// TIA Portal project "bao_cao" (V15.1)

(* hardware
DEVICE "S71500/ET200MP station_1"  S7-1500 station
   slot 0: "Rail_0"  Rack  6ES7 590-1***0-0AA0
   slot 1: "PLC_1"  CPU 1516-3 PN/DP  6ES7 516-3AN00-0AB0  V1.7
DEVICE "PC-System_1"  SIMATIC PC station
   slot 0: "SIMATIC PC station"  Rail  SIMATIC PC-Station  V1.0
      slot 125: "Stationmanager"  Station_Manager  V6.0.4
   slot 1: "HMI_RT_1"  WinCC RT Advanced  6AV2 104-0xxxx-xxxx  15.1.0.0
      slot 33792: "Host interface"  Host interface
   slot 2: "IE general_1"  IE General  IE_CP  V8.2.0
*)

// ===== PLC "PLC_1"  CPU 1516-3 PN/DP =====

VAR_GLOBAL   // PLC tag table "Default tag table"
   "Tag_1" AT %M100.0 : Bool;
END_VAR

VAR_GLOBAL   // PLC tag table "INPUT"
   "BI_START" AT %I0.0 : Bool;
   "BI_STOP" AT %I0.1 : Bool;
   "BI_AUTO" AT %I0.2 : Bool;
   "BI_MANU" AT %I0.3 : Bool;
   "I_CB1" AT %I0.4 : Bool;
   "I_CB2" AT %I0.5 : Bool;
   "I_CB3" AT %I0.6 : Bool;
   "I_CB_DAY" AT %I0.7 : Bool;
   "BM_START" AT %M0.0 : Bool;
   "BM_STOP" AT %M0.1 : Bool;
   "BM_AUTO" AT %M0.2 : Bool;
   "BM_MANU" AT %M0.3 : Bool;
   "M_CB1" AT %M0.4 : Bool;
   "M_CB2" AT %M0.5 : Bool;
   "M_CB3" AT %M0.6 : Bool;
   "M_CB_DAY" AT %M0.7 : Bool;
   "BM_SIMULATION" AT %M1.0 : Bool;
   "BIT_GIU" AT %M1.1 : Bool;
END_VAR

VAR_GLOBAL   // PLC tag table "OUTPUT"
   "Q_DEN_LV" AT %Q0.0 : Bool;
   "Q_BT" AT %Q0.1 : Bool;
   "Q_BOM_DL" AT %Q0.2 : Bool;
   "Q_XLC1" AT %Q0.3 : Bool;
   "Q_XLC2" AT %Q0.4 : Bool;
   "Q_XLK1" AT %Q0.5 : Bool;
   "Q_XLK2" AT %Q0.6 : Bool;
   "Q_XL_DAY_NAP" AT %Q0.7 : Bool;
   "Q_XL_DONG_NAP" AT %Q1.0 : Bool;
END_VAR

VAR_GLOBAL   // PLC tag table "DEM_SP"
   "DEM_CB1" AT %MW100 : Int;
   "DEM_CB2" AT %MW102 : Int;
   "DEM_CB3" AT %MW104 : Int;
END_VAR

VAR_GLOBAL   // PLC tag table "LENH_P&N"
   "P1" AT %M10.0 : Bool;
   "P2" AT %M10.1 : Bool;
   "BIT_DELAY3S_1" AT %M10.2 : Bool;
   "BIT_DELAY3S_2" AT %M10.3 : Bool;
   "BAO_DANG_ROT" AT %M10.4 : Bool;
   "BAO_DANG_DAP_NAP" AT %M10.5 : Bool;
   "BIT_DELAY3S_3" AT %M10.6 : Bool;
   "BIT_DELAY1S_1" AT %M10.7 : Bool;
   "BIT_DELAY1S_2" AT %M11.0 : Bool;
   "BIT_DELAY3S_4" AT %M11.1 : Bool;
   "BIT_DELAY3S_5" AT %M11.2 : Bool;
   "P3" AT %M11.3 : Bool;
   "P4" AT %M11.4 : Bool;
   "P5" AT %M11.5 : Bool;
   "P6" AT %M11.6 : Bool;
   "P7" AT %M11.7 : Bool;
   "P8" AT %M12.0 : Bool;
   "XUNG_1S" AT %M12.1 : Bool;
   "P10" AT %M12.2 : Bool;
   "P11" AT %M12.3 : Bool;
   "P12" AT %M12.4 : Bool;
   "P13" AT %M12.5 : Bool;
   "P14" AT %M12.6 : Bool;
   "P15" AT %M12.7 : Bool;
   "P16" AT %M13.0 : Bool;
END_VAR

VAR_GLOBAL   // PLC tag table "SIMULATION"
   "SIMU_DOAN_1" AT %MW106 : Int;
   "SIMU_DOAN_2" AT %MW108 : Int;
   "SIMU_DOAN_3" AT %MW110 : Int;
   "BIT_CHAI_MOVE_DOAN_1" AT %M20.0 : Bool;
   "BIT_CHAI_MOVE_DOAN_2" AT %M20.1 : Bool;
   "BIT_CHAI_MOVE_DOAN_3" AT %M20.2 : Bool;
   "SIMU_CHAI_DANG_DONG_NAP" AT %M20.3 : Bool;
   "SIMU_CHAI_DANG_ROT" AT %M20.4 : Bool;
END_VAR

// folder: System blocks/Program resources

DATA_BLOCK "IEC_Timer_0_DB"   // DB1
{ S7_Optimized_Access := 'TRUE' }
AUTHOR : Simatic
FAMILY : IEC
NAME : IEC_TMR
VERSION : 1.0
// stored: InstanceOfName IEC_TIMER
"IEC_TIMER"
BEGIN
END_DATA_BLOCK

DATA_BLOCK "IEC_Timer_0_DB_1"   // DB2
{ S7_Optimized_Access := 'TRUE' }
AUTHOR : Simatic
FAMILY : IEC
NAME : IEC_TMR
VERSION : 1.0
// stored: InstanceOfName IEC_TIMER
"IEC_TIMER"
BEGIN
END_DATA_BLOCK

DATA_BLOCK "IEC_Timer_0_DB_2"   // DB3
{ S7_Optimized_Access := 'TRUE' }
AUTHOR : Simatic
FAMILY : IEC
NAME : IEC_TMR
VERSION : 1.0
// stored: InstanceOfName IEC_TIMER
"IEC_TIMER"
BEGIN
END_DATA_BLOCK

DATA_BLOCK "IEC_Timer_0_DB_3"   // DB4
{ S7_Optimized_Access := 'TRUE' }
AUTHOR : Simatic
FAMILY : IEC
NAME : IEC_TMR
VERSION : 1.0
// stored: InstanceOfName IEC_TIMER
"IEC_TIMER"
BEGIN
END_DATA_BLOCK

DATA_BLOCK "IEC_Timer_0_DB_4"   // DB5
{ S7_Optimized_Access := 'TRUE' }
AUTHOR : Simatic
FAMILY : IEC
NAME : IEC_TMR
VERSION : 1.0
// stored: InstanceOfName IEC_TIMER
"IEC_TIMER"
BEGIN
END_DATA_BLOCK

DATA_BLOCK "IEC_Timer_0_DB_5"   // DB6
{ S7_Optimized_Access := 'TRUE' }
AUTHOR : Simatic
FAMILY : IEC
NAME : IEC_TMR
VERSION : 1.0
// stored: InstanceOfName IEC_TIMER
"IEC_TIMER"
BEGIN
END_DATA_BLOCK

DATA_BLOCK "IEC_Timer_0_DB_6"   // DB7
{ S7_Optimized_Access := 'TRUE' }
AUTHOR : Simatic
FAMILY : IEC
NAME : IEC_TMR
VERSION : 1.0
// stored: InstanceOfName IEC_TIMER
"IEC_TIMER"
BEGIN
END_DATA_BLOCK

DATA_BLOCK "IEC_Timer_0_DB_7"   // DB8
{ S7_Optimized_Access := 'TRUE' }
AUTHOR : Simatic
FAMILY : IEC
NAME : IEC_TMR
VERSION : 1.0
// stored: InstanceOfName IEC_TIMER
"IEC_TIMER"
BEGIN
END_DATA_BLOCK

DATA_BLOCK "IEC_Timer_0_DB_8"   // DB9
{ S7_Optimized_Access := 'TRUE' }
AUTHOR : Simatic
FAMILY : IEC
NAME : IEC_TMR
VERSION : 1.0
// stored: InstanceOfName IEC_TIMER
"IEC_TIMER"
BEGIN
END_DATA_BLOCK

DATA_BLOCK "IEC_Timer_0_DB_9"   // DB10
{ S7_Optimized_Access := 'TRUE' }
AUTHOR : Simatic
FAMILY : IEC
NAME : IEC_TMR
VERSION : 1.0
// stored: InstanceOfName IEC_TIMER
"IEC_TIMER"
BEGIN
END_DATA_BLOCK

// folder: (top level)

FUNCTION "CHE_DO_TU_DONG" : Void   // FC1, LAD
{ S7_Optimized_Access := 'TRUE' }
VERSION : 0.1
   VAR_TEMP   // added for the SCL form of the ladder/FBD networks
      _w1 : Bool;
   END_VAR
BEGIN

REGION Network 1
   // KHI ẤN NÚT AUTO THÌ BẬT BĂNG TẢI
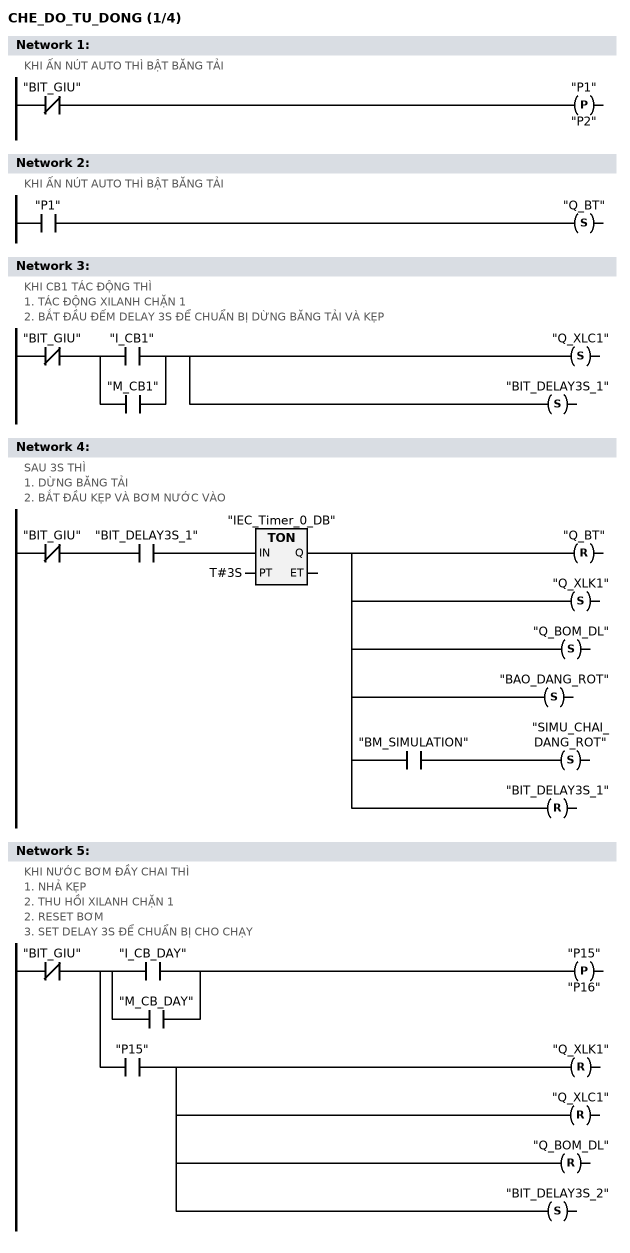
   "P1" := NOT "BIT_GIU" AND NOT "P2";   // rising edge
   "P2" := NOT "BIT_GIU";
END_REGION

REGION Network 2
   // KHI ẤN NÚT AUTO THÌ BẬT BĂNG TẢI
   RUNG wire#powerrail
      Contact( "P1" )
      S_Coil( "Q_BT" )
   END_RUNG
   // the same network as SCL:
   IF "P1" THEN "Q_BT" := TRUE; END_IF;
END_REGION

REGION Network 3
   // KHI CB1 TÁC ĐỘNG THÌ
   // 1. TÁC ĐỘNG XILANH CHẶN 1
   // 2. BẮT ĐẦU ĐẾM DELAY 3S ĐỂ CHUẨN BỊ DỪNG BĂNG TẢI VÀ KẸP
   RUNG wire#powerrail
      I_Contact( "BIT_GIU" )
      wire#w1
      Contact( "I_CB1" )
      wire#w2
      S_Coil( "Q_XLC1" )
   END_RUNG
   RUNG wire#w1
      Contact( "M_CB1" )
   END_RUNG wire#w2
   RUNG wire#w2
      S_Coil( "BIT_DELAY3S_1" )
   END_RUNG
   // the same network as SCL:
   IF NOT "BIT_GIU" AND ("I_CB1" OR "M_CB1") THEN
       "Q_XLC1" := TRUE;
       "BIT_DELAY3S_1" := TRUE;
   END_IF;
END_REGION

REGION Network 4
   // SAU 3S THÌ
   // 1. DỪNG BĂNG TẢI
   // 2. BẮT ĐẦU KẸP VÀ BƠM NƯỚC VÀO
   "IEC_Timer_0_DB".TON(IN := NOT "BIT_GIU" AND "BIT_DELAY3S_1", PT := T#3S);
   IF "IEC_Timer_0_DB".Q THEN
       "Q_BT" := FALSE;
       "Q_XLK1" := TRUE;
       "Q_BOM_DL" := TRUE;
       "BAO_DANG_ROT" := TRUE;
   END_IF;
   IF "IEC_Timer_0_DB".Q AND "BM_SIMULATION" THEN "SIMU_CHAI_DANG_ROT" := TRUE; END_IF;
   IF "IEC_Timer_0_DB".Q THEN "BIT_DELAY3S_1" := FALSE; END_IF;
END_REGION

REGION Network 5
   // KHI NƯỚC BƠM ĐẦY CHAI THÌ
   // 1. NHẢ KẸP
   // 2. THU HỒI XILANH CHẶN 1
   // 2. RESET BƠM
   // 3. SET DELAY 3S ĐỂ CHUẨN BỊ CHO CHẠY
   #_w1 := NOT "BIT_GIU" AND ("I_CB_DAY" OR "M_CB_DAY");
   "P15" := #_w1 AND NOT "P16";   // rising edge
   "P16" := #_w1;
   IF NOT "BIT_GIU" AND "P15" THEN
       "Q_XLK1" := FALSE;
       "Q_XLC1" := FALSE;
       "Q_BOM_DL" := FALSE;
       "BIT_DELAY3S_2" := TRUE;
   END_IF;
END_REGION

REGION Network 6
   // SAU 3S THÌ
   // 1. CHO BĂNG TẢI CHẠY
   // (NGOÀI RA CÒN THÊM BÍT MÔ PHỎNG CHAI DI CHUYỂN ĐOẠN 2 VÀ 1)
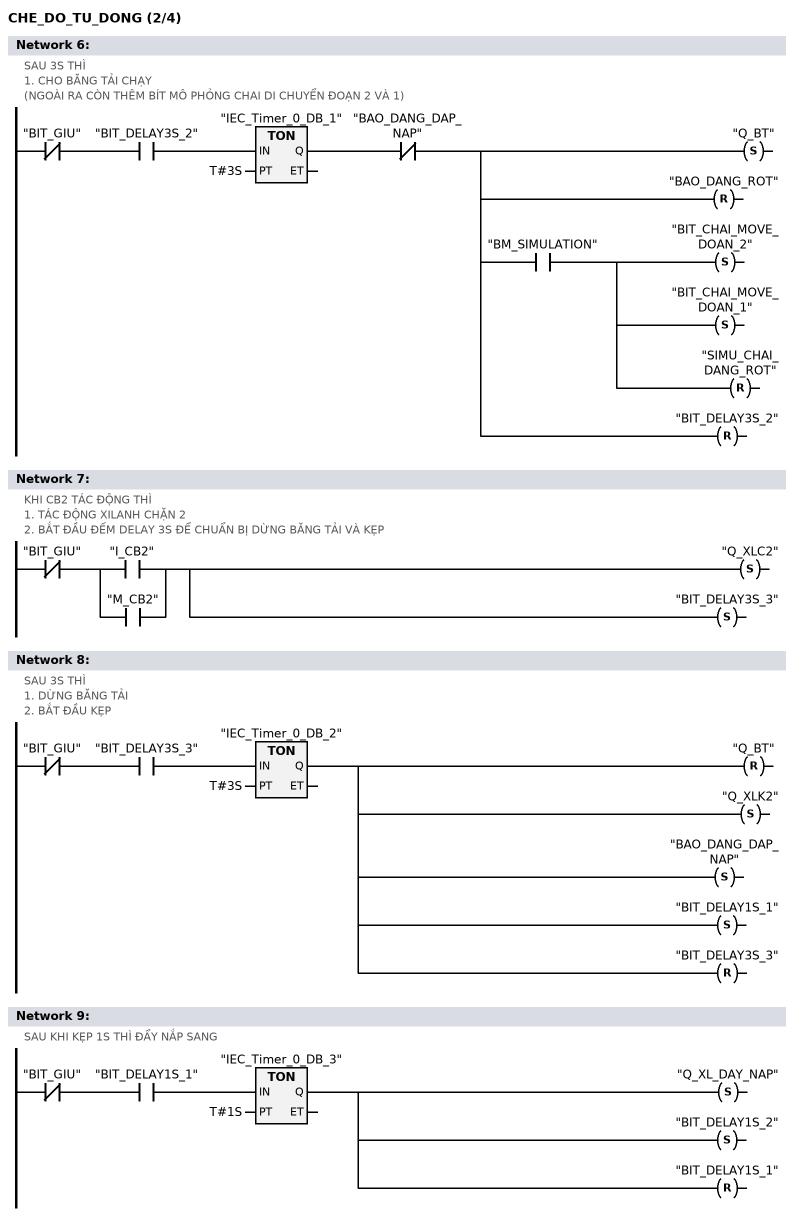
   "IEC_Timer_0_DB_1".TON(IN := NOT "BIT_GIU" AND "BIT_DELAY3S_2", PT := T#3S);
   #_w1 := "IEC_Timer_0_DB_1".Q AND NOT "BAO_DANG_DAP_NAP";
   IF #_w1 THEN
       "Q_BT" := TRUE;
       "BAO_DANG_ROT" := FALSE;
   END_IF;
   IF #_w1 AND "BM_SIMULATION" THEN
       "BIT_CHAI_MOVE_DOAN_2" := TRUE;
       "BIT_CHAI_MOVE_DOAN_1" := TRUE;
       "SIMU_CHAI_DANG_ROT" := FALSE;
   END_IF;
   IF #_w1 THEN "BIT_DELAY3S_2" := FALSE; END_IF;
END_REGION

REGION Network 7
   // KHI CB2 TÁC ĐỘNG THÌ
   // 1. TÁC ĐỘNG XILANH CHẶN 2
   // 2. BẮT ĐẦU ĐẾM DELAY 3S ĐỂ CHUẨN BỊ DỪNG BĂNG TẢI VÀ KẸP
   RUNG wire#powerrail
      I_Contact( "BIT_GIU" )
      wire#w1
      Contact( "I_CB2" )
      wire#w2
      S_Coil( "Q_XLC2" )
   END_RUNG
   RUNG wire#w1
      Contact( "M_CB2" )
   END_RUNG wire#w2
   RUNG wire#w2
      S_Coil( "BIT_DELAY3S_3" )
   END_RUNG
   // the same network as SCL:
   IF NOT "BIT_GIU" AND ("I_CB2" OR "M_CB2") THEN
       "Q_XLC2" := TRUE;
       "BIT_DELAY3S_3" := TRUE;
   END_IF;
END_REGION

REGION Network 8
   // SAU 3S THÌ
   // 1. DỪNG BĂNG TẢI
   // 2. BẮT ĐẦU KẸP
   "IEC_Timer_0_DB_2".TON(IN := NOT "BIT_GIU" AND "BIT_DELAY3S_3", PT := T#3S);
   IF "IEC_Timer_0_DB_2".Q THEN
       "Q_BT" := FALSE;
       "Q_XLK2" := TRUE;
       "BAO_DANG_DAP_NAP" := TRUE;
       "BIT_DELAY1S_1" := TRUE;
       "BIT_DELAY3S_3" := FALSE;
   END_IF;
END_REGION

REGION Network 9
   // SAU KHI KẸP 1S THÌ ĐẨY NẮP SANG
   "IEC_Timer_0_DB_3".TON(IN := NOT "BIT_GIU" AND "BIT_DELAY1S_1", PT := T#1S);
   IF "IEC_Timer_0_DB_3".Q THEN
       "Q_XL_DAY_NAP" := TRUE;
       "BIT_DELAY1S_2" := TRUE;
       "BIT_DELAY1S_1" := FALSE;
   END_IF;
END_REGION

REGION Network 10
   // SAU 1S THÌ ĐÓNG NẮP XUỐNG VÀ XL ĐẨY NẮP VỀ
   // VÀ SET DELAY 3S
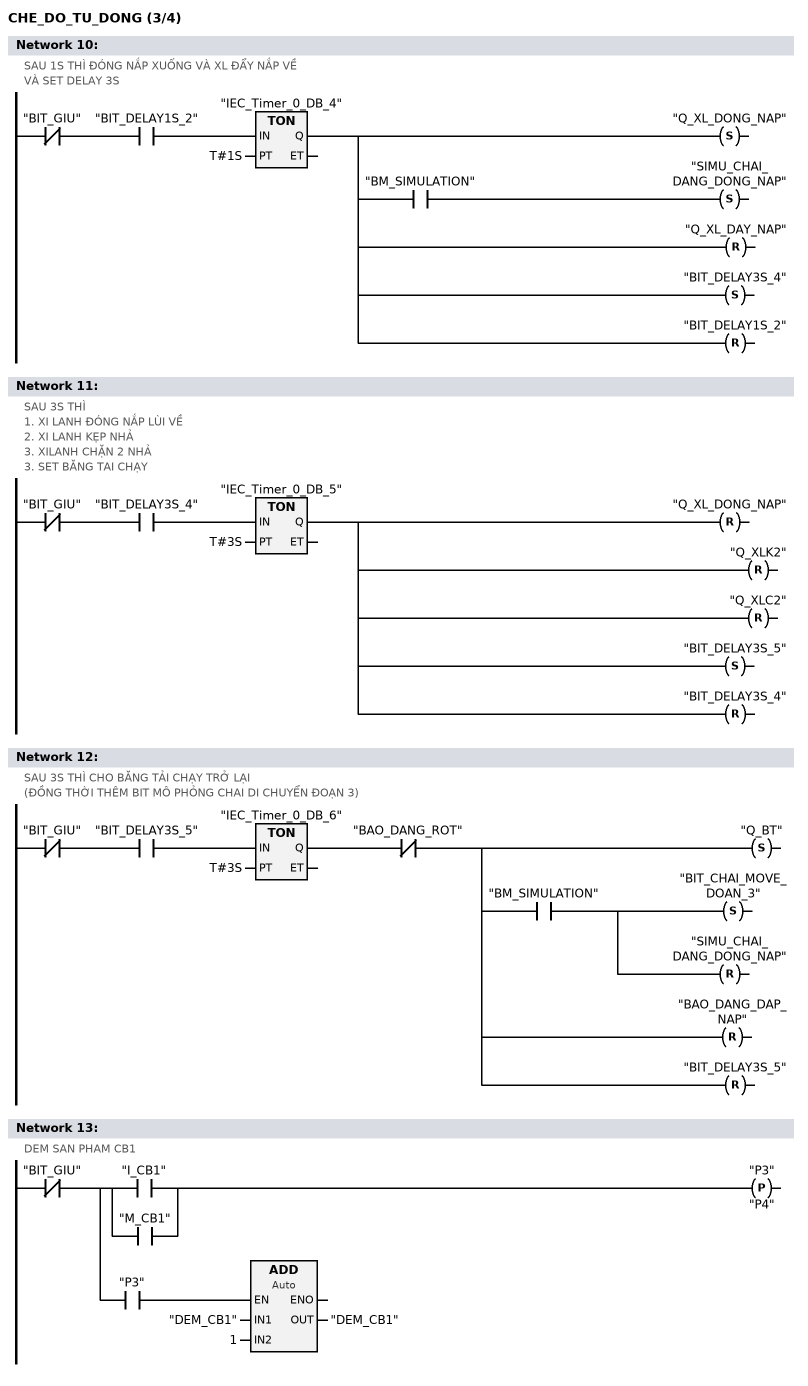
   "IEC_Timer_0_DB_4".TON(IN := NOT "BIT_GIU" AND "BIT_DELAY1S_2", PT := T#1S);
   IF "IEC_Timer_0_DB_4".Q THEN "Q_XL_DONG_NAP" := TRUE; END_IF;
   IF "IEC_Timer_0_DB_4".Q AND "BM_SIMULATION" THEN "SIMU_CHAI_DANG_DONG_NAP" := TRUE; END_IF;
   IF "IEC_Timer_0_DB_4".Q THEN
       "Q_XL_DAY_NAP" := FALSE;
       "BIT_DELAY3S_4" := TRUE;
       "BIT_DELAY1S_2" := FALSE;
   END_IF;
END_REGION

REGION Network 11
   // SAU 3S THÌ
   // 1. XI LANH ĐÓNG NẮP LÙI VỀ
   // 2. XI LANH KẸP NHẢ
   // 3. XILANH CHẶN 2 NHẢ
   // 3. SET BĂNG TAI CHẠY
   "IEC_Timer_0_DB_5".TON(IN := NOT "BIT_GIU" AND "BIT_DELAY3S_4", PT := T#3S);
   IF "IEC_Timer_0_DB_5".Q THEN
       "Q_XL_DONG_NAP" := FALSE;
       "Q_XLK2" := FALSE;
       "Q_XLC2" := FALSE;
       "BIT_DELAY3S_5" := TRUE;
       "BIT_DELAY3S_4" := FALSE;
   END_IF;
END_REGION

REGION Network 12
   // SAU 3S THÌ CHO BĂNG TẢI CHẠY TRỞ LẠI
   // (ĐỒNG THỜI THÊM BIT MÔ PHỎNG CHAI DI CHUYỂN ĐOẠN 3)
   "IEC_Timer_0_DB_6".TON(IN := NOT "BIT_GIU" AND "BIT_DELAY3S_5", PT := T#3S);
   #_w1 := "IEC_Timer_0_DB_6".Q AND NOT "BAO_DANG_ROT";
   IF #_w1 THEN "Q_BT" := TRUE; END_IF;
   IF #_w1 AND "BM_SIMULATION" THEN
       "BIT_CHAI_MOVE_DOAN_3" := TRUE;
       "SIMU_CHAI_DANG_DONG_NAP" := FALSE;
   END_IF;
   IF #_w1 THEN
       "BAO_DANG_DAP_NAP" := FALSE;
       "BIT_DELAY3S_5" := FALSE;
   END_IF;
END_REGION

REGION Network 13
   // DEM SAN PHAM CB1
   #_w1 := NOT "BIT_GIU" AND ("I_CB1" OR "M_CB1");
   "P3" := #_w1 AND NOT "P4";   // rising edge
   "P4" := #_w1;
   IF NOT "BIT_GIU" AND "P3" THEN "DEM_CB1" := "DEM_CB1" + 1; END_IF;
END_REGION

REGION Network 14
   // DEM SAN PHAM CB2
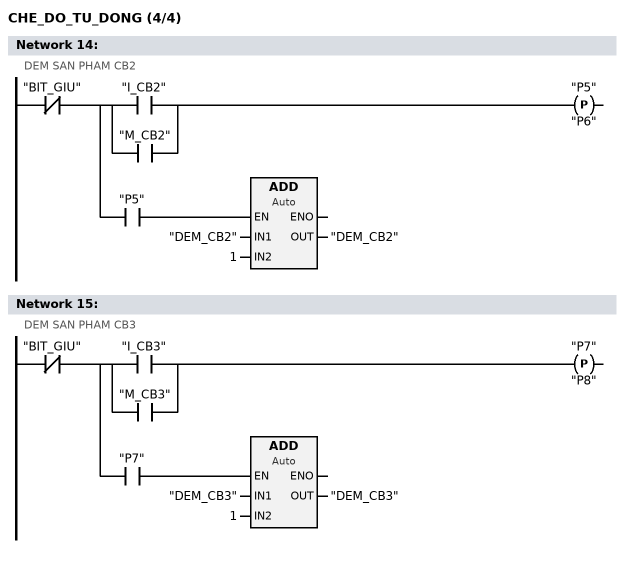
   #_w1 := NOT "BIT_GIU" AND ("I_CB2" OR "M_CB2");
   "P5" := #_w1 AND NOT "P6";   // rising edge
   "P6" := #_w1;
   IF NOT "BIT_GIU" AND "P5" THEN "DEM_CB2" := "DEM_CB2" + 1; END_IF;
END_REGION

REGION Network 15
   // DEM SAN PHAM CB3
   #_w1 := NOT "BIT_GIU" AND ("I_CB3" OR "M_CB3");
   "P7" := #_w1 AND NOT "P8";   // rising edge
   "P8" := #_w1;
   IF NOT "BIT_GIU" AND "P7" THEN "DEM_CB3" := "DEM_CB3" + 1; END_IF;
END_REGION
END_FUNCTION

FUNCTION "CHE_DO_BANG_TAY" : Void   // FC2, LAD
{ S7_Optimized_Access := 'TRUE' }
VERSION : 0.1
BEGIN
END_FUNCTION

FUNCTION "KHOI_MO_PHONG" : Void   // FC3, LAD
{ S7_Optimized_Access := 'TRUE' }
VERSION : 0.1
   VAR_TEMP   // added for the SCL form of the ladder/FBD networks
      _w1 : Bool;
   END_VAR
BEGIN

REGION Network 1
   // TAO TIMER DEM 1S TAC DONG 1 LAN
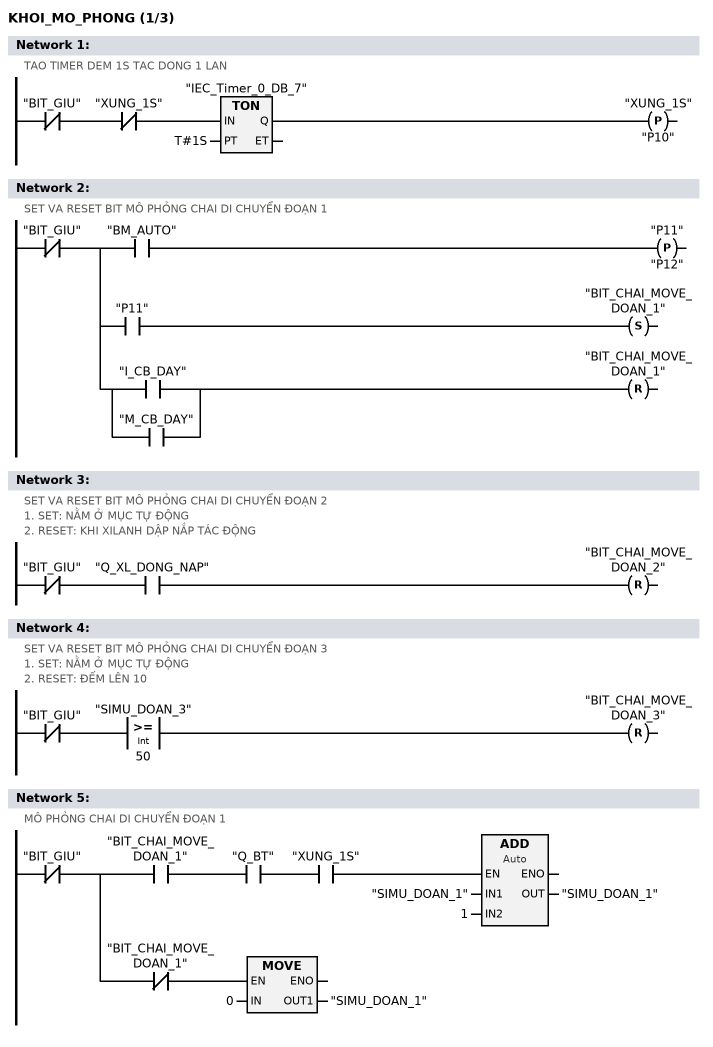
   "IEC_Timer_0_DB_7".TON(IN := NOT "BIT_GIU" AND NOT "XUNG_1S", PT := T#1S);
   "XUNG_1S" := "IEC_Timer_0_DB_7".Q AND NOT "P10";   // rising edge
   "P10" := "IEC_Timer_0_DB_7".Q;
END_REGION

REGION Network 2
   // SET VA RESET BIT MÔ PHỎNG CHAI DI CHUYỂN ĐOẠN 1
   #_w1 := NOT "BIT_GIU" AND "BM_AUTO";
   "P11" := #_w1 AND NOT "P12";   // rising edge
   "P12" := #_w1;
   IF NOT "BIT_GIU" AND "P11" THEN "BIT_CHAI_MOVE_DOAN_1" := TRUE; END_IF;
   IF NOT "BIT_GIU" AND ("I_CB_DAY" OR "M_CB_DAY") THEN "BIT_CHAI_MOVE_DOAN_1" := FALSE; END_IF;
END_REGION

REGION Network 3
   // SET VA RESET BIT MÔ PHỎNG CHAI DI CHUYỂN ĐOẠN 2
   // 1. SET: NẰM Ở MỤC TỰ ĐỘNG
   // 2. RESET: KHI XILANH DẬP NẮP TÁC ĐỘNG
   RUNG wire#powerrail
      I_Contact( "BIT_GIU" )
      Contact( "Q_XL_DONG_NAP" )
      R_Coil( "BIT_CHAI_MOVE_DOAN_2" )
   END_RUNG
   // the same network as SCL:
   IF NOT "BIT_GIU" AND "Q_XL_DONG_NAP" THEN "BIT_CHAI_MOVE_DOAN_2" := FALSE; END_IF;
END_REGION

REGION Network 4
   // SET VA RESET BIT MÔ PHỎNG CHAI DI CHUYỂN ĐOẠN 3
   // 1. SET: NẰM Ở MỤC TỰ ĐỘNG
   // 2. RESET: ĐẾM LÊN 10
   RUNG wire#powerrail
      I_Contact( "BIT_GIU" )
      { S7_Templates := "SrcType := Int" } GE_Contact(in1 := "SIMU_DOAN_3", in2 := 50)
      R_Coil( "BIT_CHAI_MOVE_DOAN_3" )
   END_RUNG
   // the same network as SCL:
   IF NOT "BIT_GIU" AND ("SIMU_DOAN_3" >= 50) THEN "BIT_CHAI_MOVE_DOAN_3" := FALSE; END_IF;
END_REGION

REGION Network 5
   // MÔ PHỎNG CHAI DI CHUYỂN ĐOẠN 1
   RUNG wire#powerrail
      I_Contact( "BIT_GIU" )
      wire#w1
      Contact( "BIT_CHAI_MOVE_DOAN_1" )
      Contact( "Q_BT" )
      Contact( "XUNG_1S" )
      Add(in1 := "SIMU_DOAN_1", in2 := 1, out => "SIMU_DOAN_1")
   END_RUNG
   RUNG wire#w1
      I_Contact( "BIT_CHAI_MOVE_DOAN_1" )
      Move(in := 0, out1 => "SIMU_DOAN_1")
   END_RUNG
   // the same network as SCL:
   IF NOT "BIT_GIU" AND "BIT_CHAI_MOVE_DOAN_1" AND "Q_BT" AND "XUNG_1S" THEN
       "SIMU_DOAN_1" := "SIMU_DOAN_1" + 1;
   END_IF;
   IF NOT "BIT_GIU" AND NOT "BIT_CHAI_MOVE_DOAN_1" THEN "SIMU_DOAN_1" := 0; END_IF;
END_REGION

REGION Network 6
   // MÔ PHỎNG CHAI DI CHUYỂN ĐOẠN 2
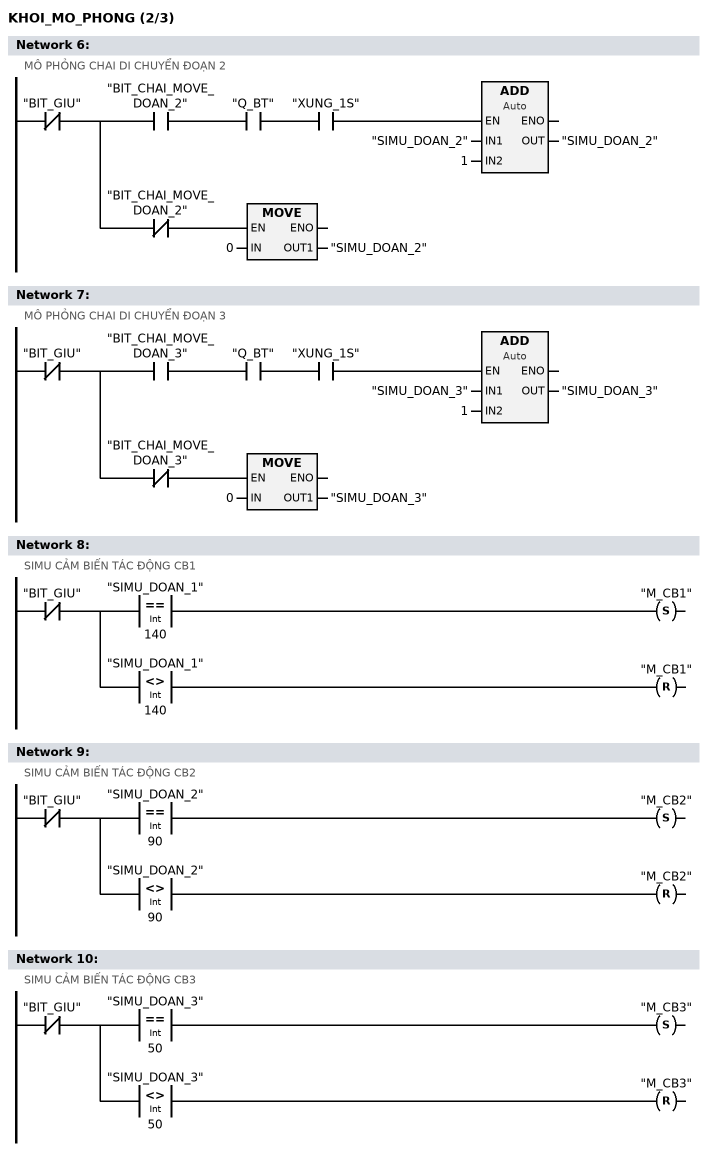
   RUNG wire#powerrail
      I_Contact( "BIT_GIU" )
      wire#w1
      Contact( "BIT_CHAI_MOVE_DOAN_2" )
      Contact( "Q_BT" )
      Contact( "XUNG_1S" )
      Add(in1 := "SIMU_DOAN_2", in2 := 1, out => "SIMU_DOAN_2")
   END_RUNG
   RUNG wire#w1
      I_Contact( "BIT_CHAI_MOVE_DOAN_2" )
      Move(in := 0, out1 => "SIMU_DOAN_2")
   END_RUNG
   // the same network as SCL:
   IF NOT "BIT_GIU" AND "BIT_CHAI_MOVE_DOAN_2" AND "Q_BT" AND "XUNG_1S" THEN
       "SIMU_DOAN_2" := "SIMU_DOAN_2" + 1;
   END_IF;
   IF NOT "BIT_GIU" AND NOT "BIT_CHAI_MOVE_DOAN_2" THEN "SIMU_DOAN_2" := 0; END_IF;
END_REGION

REGION Network 7
   // MÔ PHỎNG CHAI DI CHUYỂN ĐOẠN 3
   RUNG wire#powerrail
      I_Contact( "BIT_GIU" )
      wire#w1
      Contact( "BIT_CHAI_MOVE_DOAN_3" )
      Contact( "Q_BT" )
      Contact( "XUNG_1S" )
      Add(in1 := "SIMU_DOAN_3", in2 := 1, out => "SIMU_DOAN_3")
   END_RUNG
   RUNG wire#w1
      I_Contact( "BIT_CHAI_MOVE_DOAN_3" )
      Move(in := 0, out1 => "SIMU_DOAN_3")
   END_RUNG
   // the same network as SCL:
   IF NOT "BIT_GIU" AND "BIT_CHAI_MOVE_DOAN_3" AND "Q_BT" AND "XUNG_1S" THEN
       "SIMU_DOAN_3" := "SIMU_DOAN_3" + 1;
   END_IF;
   IF NOT "BIT_GIU" AND NOT "BIT_CHAI_MOVE_DOAN_3" THEN "SIMU_DOAN_3" := 0; END_IF;
END_REGION

REGION Network 8
   // SIMU CẢM BIẾN TÁC ĐỘNG CB1
   RUNG wire#powerrail
      I_Contact( "BIT_GIU" )
      wire#w1
      { S7_Templates := "SrcType := Int" } EQ_Contact(in1 := "SIMU_DOAN_1", in2 := 140)
      S_Coil( "M_CB1" )
   END_RUNG
   RUNG wire#w1
      { S7_Templates := "SrcType := Int" } NE_Contact(in1 := "SIMU_DOAN_1", in2 := 140)
      R_Coil( "M_CB1" )
   END_RUNG
   // the same network as SCL:
   IF NOT "BIT_GIU" AND ("SIMU_DOAN_1" = 140) THEN "M_CB1" := TRUE; END_IF;
   IF NOT "BIT_GIU" AND ("SIMU_DOAN_1" <> 140) THEN "M_CB1" := FALSE; END_IF;
END_REGION

REGION Network 9
   // SIMU CẢM BIẾN TÁC ĐỘNG CB2
   RUNG wire#powerrail
      I_Contact( "BIT_GIU" )
      wire#w1
      { S7_Templates := "SrcType := Int" } EQ_Contact(in1 := "SIMU_DOAN_2", in2 := 90)
      S_Coil( "M_CB2" )
   END_RUNG
   RUNG wire#w1
      { S7_Templates := "SrcType := Int" } NE_Contact(in1 := "SIMU_DOAN_2", in2 := 90)
      R_Coil( "M_CB2" )
   END_RUNG
   // the same network as SCL:
   IF NOT "BIT_GIU" AND ("SIMU_DOAN_2" = 90) THEN "M_CB2" := TRUE; END_IF;
   IF NOT "BIT_GIU" AND ("SIMU_DOAN_2" <> 90) THEN "M_CB2" := FALSE; END_IF;
END_REGION

REGION Network 10
   // SIMU CẢM BIẾN TÁC ĐỘNG CB3
   RUNG wire#powerrail
      I_Contact( "BIT_GIU" )
      wire#w1
      { S7_Templates := "SrcType := Int" } EQ_Contact(in1 := "SIMU_DOAN_3", in2 := 50)
      S_Coil( "M_CB3" )
   END_RUNG
   RUNG wire#w1
      { S7_Templates := "SrcType := Int" } NE_Contact(in1 := "SIMU_DOAN_3", in2 := 50)
      R_Coil( "M_CB3" )
   END_RUNG
   // the same network as SCL:
   IF NOT "BIT_GIU" AND ("SIMU_DOAN_3" = 50) THEN "M_CB3" := TRUE; END_IF;
   IF NOT "BIT_GIU" AND ("SIMU_DOAN_3" <> 50) THEN "M_CB3" := FALSE; END_IF;
END_REGION

REGION Network 11
   // TÁC ĐỘNG CẢM BIẾN ĐẦY SAU KHI ĐỘNG CƠ RÓT 5S SAU 3S THÌ RESET CB ĐẦY
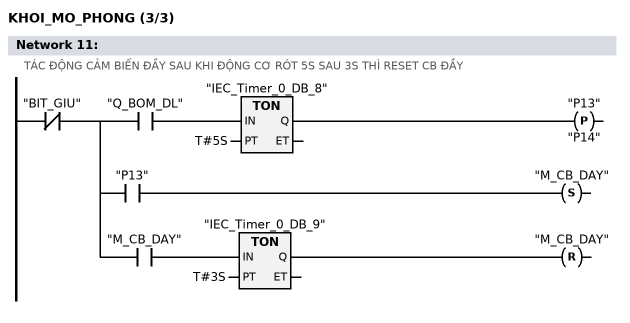
   "IEC_Timer_0_DB_8".TON(IN := NOT "BIT_GIU" AND "Q_BOM_DL", PT := T#5S);
   "P13" := "IEC_Timer_0_DB_8".Q AND NOT "P14";   // rising edge
   "P14" := "IEC_Timer_0_DB_8".Q;
   IF NOT "BIT_GIU" AND "P13" THEN "M_CB_DAY" := TRUE; END_IF;
   "IEC_Timer_0_DB_9".TON(IN := NOT "BIT_GIU" AND "M_CB_DAY", PT := T#3S);
   IF "IEC_Timer_0_DB_9".Q THEN "M_CB_DAY" := FALSE; END_IF;
END_REGION
END_FUNCTION

ORGANIZATION_BLOCK "Main"   // OB1, LAD, ProgramCycle
TITLE = "Main Program Sweep (Cycle)"
{ S7_Optimized_Access := 'TRUE' }
VERSION : 0.1
   VAR_INPUT
      Initial_Call : Bool;   // Initial call of this OB
      Remanence : Bool;   // =True, if remanent data are available
   END_VAR
   VAR_TEMP   // added for the SCL form of the ladder/FBD networks
      _w1 : Bool;
   END_VAR
BEGIN

REGION Network 1
   // KHỎI ĐỘNG HỆ THỐNG
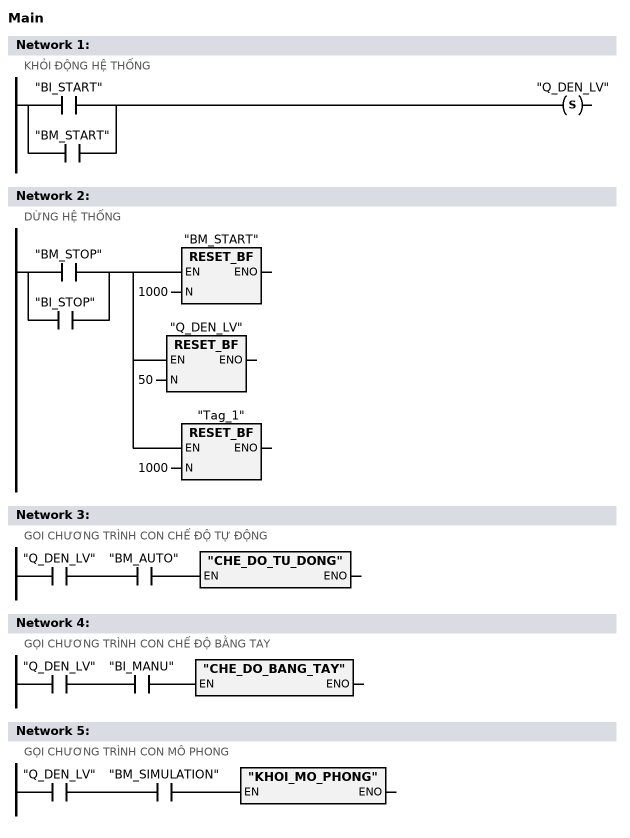
   RUNG wire#powerrail
      Contact( "BI_START" )
      wire#w1
      S_Coil( "Q_DEN_LV" )
   END_RUNG
   RUNG wire#powerrail
      Contact( "BM_START" )
   END_RUNG wire#w1
   // the same network as SCL:
   IF "BI_START" OR "BM_START" THEN "Q_DEN_LV" := TRUE; END_IF;
END_REGION

REGION Network 2
   // DỪNG HỆ THỐNG
   // no SCL statement known for RBitfield: written as a call
   #_w1 := "BM_STOP" OR "BI_STOP";
   IF #_w1 THEN
       RESET_BF(operand := "BM_START", n := 1000);
       RESET_BF(operand := "Q_DEN_LV", n := 50);
       RESET_BF(operand := "Tag_1", n := 1000);
   END_IF;
END_REGION

REGION Network 3
   // GOI CHƯƠNG TRÌNH CON CHẾ ĐỘ TỰ ĐỘNG
   RUNG wire#powerrail
      Contact( "Q_DEN_LV" )
      Contact( "BM_AUTO" )
      "CHE_DO_TU_DONG"()
   END_RUNG
   // the same network as SCL:
   IF "Q_DEN_LV" AND "BM_AUTO" THEN "CHE_DO_TU_DONG"(); END_IF;
END_REGION

REGION Network 4
   // GỌI CHƯƠNG TRÌNH CON CHẾ ĐỘ BẰNG TAY
   RUNG wire#powerrail
      Contact( "Q_DEN_LV" )
      Contact( "BI_MANU" )
      "CHE_DO_BANG_TAY"()
   END_RUNG
   // the same network as SCL:
   IF "Q_DEN_LV" AND "BI_MANU" THEN "CHE_DO_BANG_TAY"(); END_IF;
END_REGION

REGION Network 5
   // GỌI CHƯƠNG TRÌNH CON MÔ PHONG
   RUNG wire#powerrail
      Contact( "Q_DEN_LV" )
      Contact( "BM_SIMULATION" )
      "KHOI_MO_PHONG"()
   END_RUNG
   // the same network as SCL:
   IF "Q_DEN_LV" AND "BM_SIMULATION" THEN "KHOI_MO_PHONG"(); END_IF;
END_REGION
END_ORGANIZATION_BLOCK

(* ===== HMI "HMI_RT_1" =====
system functions are stored by id; their names below are inferred from use
connection "HMI_Connection_1": ETHERNET, S7_1500_OMS

HMI tags "Default tag table"
   "Q_BOM_DL" : Bool = PLC Q_BOM_DL AT %Q0.2, 1 s
   "Q_XLK1" : Bool = PLC Q_XLK1 AT %Q0.5, 1 s
   "Q_XLK2" : Bool = PLC Q_XLK2 AT %Q0.6, 1 s
   "Q_XL_DONG_NAP" : Bool = PLC Q_XL_DONG_NAP AT %Q1.0, 1 s
   "Q_XLC1" : Bool = PLC Q_XLC1 AT %Q0.3, 1 s
   "Q_XLC2" : Bool = PLC Q_XLC2 AT %Q0.4, 1 s
   "M_CB_DAY" : Bool = PLC M_CB_DAY AT %M0.7, 1 s
   "M_CB1" : Bool = PLC M_CB1 AT %M0.4, 1 s
   "M_CB2" : Bool = PLC M_CB2 AT %M0.5, 1 s
   "M_CB3" : Bool = PLC M_CB3 AT %M0.6, 1 s
   "Q_XL_DAY_NAP" : Bool = PLC Q_XL_DAY_NAP AT %Q0.7, 1 s
   "BIT_CHAI_MOVE_DOAN_3" : Bool = PLC BIT_CHAI_MOVE_DOAN_3 AT %M20.2, 1 s
   "SIMU_DOAN_3" : Int = PLC SIMU_DOAN_3 AT %MW110, 1 s
   "SIMU_DOAN_1" : Int = PLC SIMU_DOAN_1 AT %MW106, 1 s
   "BIT_CHAI_MOVE_DOAN_1" : Bool = PLC BIT_CHAI_MOVE_DOAN_1 AT %M20.0, 1 s
   "BIT_CHAI_MOVE_DOAN_2" : Bool = PLC BIT_CHAI_MOVE_DOAN_2 AT %M20.1, 1 s
   "SIMU_DOAN_2" : Int = PLC SIMU_DOAN_2 AT %MW108, 1 s
   "Q_BT" : Bool = PLC Q_BT AT %Q0.1, 1 s
   "DEM_CB1" : Int = PLC DEM_CB1 AT %MW100, 1 s
   "DEM_CB2" : Int = PLC DEM_CB2 AT %MW102, 1 s
   "DEM_CB3" : Int = PLC DEM_CB3 AT %MW104, 1 s
   "Q_DEN_LV" : Bool = PLC Q_DEN_LV AT %Q0.0, 1 s
   "BM_SIMULATION" : Bool = PLC BM_SIMULATION AT %M1.0, 1 s
   "BM_AUTO" : Bool = PLC BM_AUTO AT %M0.2, 1 s
   "BM_MANU" : Bool = PLC BM_MANU AT %M0.3, 1 s
   "BM_START" : Bool = PLC BM_START AT %M0.0, 1 s
   "BM_STOP" : Bool = PLC BM_STOP AT %M0.1, 1 s
   "SIMU_CHAI_DANG_ROT" : Bool = PLC SIMU_CHAI_DANG_ROT AT %M20.4, 1 s
   "SIMU_CHAI_DANG_DONG_NAP" : Bool = PLC SIMU_CHAI_DANG_DONG_NAP AT %M20.3, 1 s

Template "Tittle" 1366x768
   TextField "Template_Text field_1" at 211,22 size 964x59; Text 'ĐIỀU KHIỂN HỆ THỐNG CHIẾT RÓT VÀ DẬP NẮP SẢN PHẨM'

screen "BANG_TAY" 1366x768, template "Tittle"
   SymbolLibrary "Symbol library_1" at 58,420 size 333x60
      Appearance <- "Q_BT"
   SymbolLibrary "Symbol library_2" at 304,420 size 333x60
      Appearance <- "Q_BT"
   SymbolLibrary "Symbol library_3" at 532,420 size 333x60
      Appearance <- "Q_BT"
   SymbolLibrary "Symbol library_4" at 741,420 size 333x60
      Appearance <- "Q_BT"
   SymbolLibrary "Symbol library_5" at 159,501 size 90x62
      Appearance <- "Q_BT"
   SymbolLibrary "Symbol library_6" at 458,426 size 32x123
      Visibility <- "Q_XLC1"
   SymbolLibrary "Symbol library_7" at 395,461 size 29x65
      Appearance <- "M_CB1"
   SymbolLibrary "Symbol library_8" at 459,480 size 30x69
      Visibility <- "Q_XLC1"
   Rectangle "Rectangle_1" at 389,362 size 32x23
      Visibility <- "Q_XLK1"
   Rectangle "Rectangle_2" at 463,362 size 32x23
      Visibility <- "Q_XLK1"
   SymbolLibrary "Symbol library_9" at 181,108 size 79x89
   Polyline "Polyline_1" at 340,165 size 99x188
      Appearance <- "Q_BOM_DL"
   SymbolLibrary "Symbol library_11" at 313,194 size 90x62
      Appearance <- "Q_BOM_DL"
   Polyline "Polyline_2" at 219,191 size 93x36
      Appearance <- "Q_BOM_DL"
   SymbolLibrary "Symbol library_12" at 757,425 size 32x123
      Visibility <- "Q_XLC2"
   SymbolLibrary "Symbol library_13" at 689,460 size 29x65
      Appearance <- "M_CB2"
   SymbolLibrary "Symbol library_14" at 758,479 size 30x69
      Visibility <- "Q_XLC2"
   Rectangle "Rectangle_3" at 688,361 size 32x23
      Visibility <- "Q_XLK2"
   Rectangle "Rectangle_4" at 762,361 size 32x23
      Visibility <- "Q_XLK2"
   SymbolLibrary "Symbol library_16" at 724,224 size 32x123
      Visibility <- "Q_XL_DONG_NAP"
   Rectangle "Rectangle_12" at 784,297 size 37x18
      Visibility <- "Q_XL_DAY_NAP"
   SymbolLibrary "Symbol library_15" at 725,224 size 30x69
      Visibility <- "Q_XL_DONG_NAP"
   Button "Button_1" at 1152,158 size 88x40; TextOff 'START'
      on Release: ResetBit("BM_START")
      on Press: SetBit("BM_START")
      Appearance <- "Q_DEN_LV"
   Button "Button_2" at 1261,158 size 88x40; TextOff 'STOP'
      on Release: ResetBit("BM_STOP")
      on Press: SetBit("BM_STOP")
      Appearance <- "Q_DEN_LV"
   Button "Button_3" at 1152,204 size 88x40; TextOff 'AUTO'
      on Press: SetBit("BM_AUTO"); ResetBit("BM_MANU"); ActivateScreen("TU_DONG", 0)
      Appearance <- "BM_AUTO"
   Button "Button_4" at 1261,204 size 88x40; TextOff 'MANU'
      on Press: SetBit("BM_MANU"); ResetBit("BM_AUTO")
      Appearance <- "BM_MANU"
   IOField "I/O field_3" at 360,556 size 75x36; FormatPattern s99999
      ProcessValue <- "DEM_CB1"
   IOField "I/O field_4" at 662,552 size 75x36; FormatPattern s99999
      ProcessValue <- "DEM_CB2"
   SymbolLibrary "Symbol library_20" at 349,340 size 45x26
      Appearance <- "M_CB_DAY"
   SymbolLibrary "Symbol library_21" at 939,457 size 29x65
      Appearance <- "M_CB3"
   TextField "Text field_17" at 1149,484 size 56x27; Text 'CB 1:'
   TextField "Text field_18" at 1293,484 size 47x27; Text '[SP]'
   IOField "I/O field_1" at 1209,481 size 84x37; FormatPattern s99999
      ProcessValue <- "DEM_CB1"
   TextField "Text field_19" at 1149,526 size 56x27; Text 'CB 2:'
   TextField "Text field_21" at 1293,526 size 47x27; Text '[SP]'
   IOField "I/O field_2" at 1209,523 size 84x37; FormatPattern s99999
      ProcessValue <- "DEM_CB2"
   TextField "Text field_22" at 1149,568 size 56x27; Text 'CB 3:'
   TextField "Text field_23" at 1293,568 size 47x27; Text '[SP]'
   IOField "I/O field_5" at 1209,565 size 84x37; FormatPattern s99999
      ProcessValue <- "DEM_CB3"
   IOField "I/O field_6" at 913,551 size 75x36; FormatPattern s99999
      ProcessValue <- "DEM_CB3"
   Button "Button_5" at 1152,322 size 88x40; TextOff 'ON'
      on Press: SetBit("BM_SIMULATION")
      Appearance <- "BM_SIMULATION"
   Button "Button_7" at 1152,368 size 88x40; TextOff 'OFF'
      on Press: ResetBit("BM_SIMULATION")
   TextField "Text field_26" at 1270,328 size 59x20; Text 'ĐÈN RUN'
   Circle "Circle_2" at 1275,352 size 49x49
      Appearance <- "Q_DEN_LV"
   SymbolLibrary "Symbol library_19" at 920,661 size 109x52
   SymbolLibrary "Symbol library_22" at 552,661 size 109x52
   SymbolLibrary "Symbol library_23" at 152,661 size 109x45
   Button "Button_6" at 1134,620 size 225x41; TextOff 'EXIT RUNTIME'
      on Press: StopRuntime(0)
   Group "Group_2" at 397,365 size 85x23
   Group "Group_3" at 695,363 size 85x23
   Group "Group_4" at 757,294 size 92x21
   Rectangle "Rectangle_8" at 722,298 size 37x18
      Visibility <- "Q_XL_DAY_NAP"
   Group "Group_5" at 832,296 size 92x21
   Button "Button_8" at 452,174 size 42x23; TextOff 'ON'
      on Press: SetBit("Q_BOM_DL")
   Button "Button_9" at 451,199 size 42x23; TextOff 'OFF'
      on Press: ResetBit("Q_BOM_DL")
   Button "Button_10" at 939,286 size 42x23; TextOff 'ON'
      on Press: SetBit("Q_XL_DAY_NAP")
   Button "Button_11" at 938,311 size 42x23; TextOff 'OFF'
      on Press: ResetBit("Q_XL_DAY_NAP")
   Button "Button_12" at 667,236 size 42x23; TextOff 'ON'
      on Press: SetBit("Q_XL_DONG_NAP")
   Button "Button_13" at 666,261 size 42x23; TextOff 'OFF'
      on Press: ResetBit("Q_XL_DONG_NAP")
   Button "Button_14" at 533,341 size 42x23; TextOff 'ON'
      on Press: SetBit("Q_XLK1")
   Button "Button_15" at 532,366 size 42x23; TextOff 'OFF'
      on Press: ResetBit("Q_XLK1")
   Button "Button_16" at 865,350 size 42x23; TextOff 'ON'
      on Press: SetBit("Q_XLK2")
   Button "Button_17" at 864,375 size 42x23; TextOff 'OFF'
      on Press: ResetBit("Q_XLK2")
   Button "Button_18" at 803,494 size 42x23; TextOff 'ON'
      on Press: SetBit("Q_XLC2")
   Button "Button_19" at 802,519 size 42x23; TextOff 'OFF'
      on Press: ResetBit("Q_XLC2")
   Button "Button_20" at 495,491 size 42x23; TextOff 'ON'
      on Press: SetBit("Q_XLC1")
   Button "Button_21" at 494,516 size 42x23; TextOff 'OFF'
      on Press: ResetBit("Q_XLC1")
   Button "Button_22" at 106,511 size 42x23; TextOff 'ON'
      on Press: SetBit("Q_BT")
   Button "Button_23" at 105,536 size 42x23; TextOff 'OFF'
      on Press: ResetBit("Q_BT")
   TextField "Text field_1" at 123,562 size 205x20; Text 'ĐỘNG CƠ BĂNG CHUYỀN'
   TextField "Text field_2" at 435,551 size 149x20; Text 'XL CHẶN CHAI 1'
   TextField "Text field_3" at 457,572 size 84x20; Text 'XL_CC_1'
   TextField "Text field_4" at 388,526 size 68x22; Text 'CB_1'
   TextField "Text field_5" at 452,301 size 102x20; Text 'XL KẸP 1'
   TextField "Text field_6" at 275,255 size 156x20; Text 'BƠM ĐỊNH LƯỢNG'
   TextField "Text field_7" at 311,278 size 94x20; Text '100ML/S'
   TextField "Text field_8" at 60,190 size 137x20; Text 'BỂ NGUYÊN LIỆU'
   TextField "Text field_9" at 736,550 size 149x20; Text 'XL CHẶN CHAI 2'
   TextField "Text field_10" at 758,571 size 84x20; Text 'XL_CC_2'
   TextField "Text field_11" at 682,525 size 68x22; Text 'CB_2'
   TextField "Text field_12" at 761,339 size 102x20; Text 'XL KẸP 2'
   TextField "Text field_13" at 856,270 size 115x20; Text 'XL ĐẨY NẮP'
   TextField "Text field_20" at 320,319 size 85x20; Text 'CB ĐẦY'
   TextField "Text field_16" at 932,522 size 75x22; Text 'CB_3'
   TextField "Text field_24" at 675,195 size 113x20; Text 'XL DẬP NẮP'
   TextField "Text field_14" at 1156,107 size 195x23; Text 'BẢNG ĐIỂU KHIỂN'
   TextField "Text field_15" at 1169,435 size 174x23; Text 'ĐẾM SẢN PHẨM'
   TextField "Text field_25" at 1150,271 size 202x23; Text 'CHẾ ĐỘ MÔ PHỎNG'
   Rectangle "Rectangle_25" at 397,365 size 32x23
      Visibility <- "Q_XLK1"
   Rectangle "Rectangle_26" at 450,365 size 32x23
      Visibility <- "Q_XLK1"
   Rectangle "Rectangle_27" at 695,363 size 32x23
      Visibility <- "Q_XLK2"
   Rectangle "Rectangle_28" at 748,363 size 32x23
      Visibility <- "Q_XLK2"
   Rectangle "Rectangle_29" at 757,294 size 23x21
      Visibility <- "Q_XL_DAY_NAP"
   Rectangle "Rectangle_30" at 779,298 size 70x14
      Visibility <- "Q_XL_DAY_NAP"
   Rectangle "Rectangle_9" at 832,296 size 23x21
      Visibility <- "Q_XL_DAY_NAP"
   Rectangle "Rectangle_31" at 854,300 size 70x14
      Visibility <- "Q_XL_DAY_NAP"

screen "TU_DONG" 1366x768, template "Tittle"
   SymbolLibrary "Symbol library_1" at 58,420 size 333x60
      Appearance <- "Q_BT"
   SymbolLibrary "Symbol library_2" at 304,420 size 333x60
      Appearance <- "Q_BT"
   SymbolLibrary "Symbol library_3" at 532,420 size 333x60
      Appearance <- "Q_BT"
   SymbolLibrary "Symbol library_4" at 741,420 size 333x60
      Appearance <- "Q_BT"
   SymbolLibrary "Symbol library_5" at 159,501 size 90x62
      Appearance <- "Q_BT"
   SymbolLibrary "Symbol library_6" at 458,426 size 32x123
      Visibility <- "Q_XLC1"
   SymbolLibrary "Symbol library_8" at 459,480 size 30x69
      Visibility <- "Q_XLC1"
   Rectangle "Rectangle_1" at 389,362 size 32x23
      Visibility <- "Q_XLK1"
   Rectangle "Rectangle_2" at 463,362 size 32x23
      Visibility <- "Q_XLK1"
   SymbolLibrary "Symbol library_9" at 181,108 size 79x89
   SymbolLibrary "Symbol library_10" at 93,353 size 39x92
      Visibility <- "BIT_CHAI_MOVE_DOAN_1"
      HorizontalMovement <- "SIMU_DOAN_1"
   Polyline "Polyline_1" at 340,165 size 99x188
      Appearance <- "Q_BOM_DL"
   SymbolLibrary "Symbol library_11" at 313,194 size 90x62
      Appearance <- "Q_BOM_DL"
   Polyline "Polyline_2" at 219,191 size 93x36
      Appearance <- "Q_BOM_DL"
   SymbolLibrary "Symbol library_12" at 757,425 size 32x123
      Visibility <- "Q_XLC2"
   SymbolLibrary "Symbol library_13" at 689,460 size 29x65
      Appearance <- "M_CB2"
   SymbolLibrary "Symbol library_14" at 758,479 size 30x69
      Visibility <- "Q_XLC2"
   Rectangle "Rectangle_3" at 688,361 size 32x23
      Visibility <- "Q_XLK2"
   Rectangle "Rectangle_4" at 762,361 size 32x23
      Visibility <- "Q_XLK2"
   SymbolLibrary "Symbol library_16" at 724,224 size 32x123
      Visibility <- "Q_XL_DONG_NAP"
   Rectangle "Rectangle_12" at 784,297 size 37x18
      Visibility <- "Q_XL_DAY_NAP"
   SymbolLibrary "Symbol library_15" at 725,224 size 30x69
      Visibility <- "Q_XL_DONG_NAP"
   Button "Button_1" at 1152,158 size 88x40; TextOff 'START'
      on Release: ResetBit("BM_START")
      on Press: SetBit("BM_START")
      Appearance <- "Q_DEN_LV"
   Button "Button_2" at 1261,158 size 88x40; TextOff 'STOP'
      on Release: ResetBit("BM_STOP")
      on Press: SetBit("BM_STOP")
      Appearance <- "Q_DEN_LV"
   Button "Button_3" at 1152,204 size 88x40; TextOff 'AUTO'
      on Press: SetBit("BM_AUTO"); ResetBit("BM_MANU")
      Appearance <- "BM_AUTO"
   Button "Button_4" at 1261,204 size 88x40; TextOff 'MANU'
      on Press: SetBit("BM_MANU"); ResetBit("BM_AUTO"); ActivateScreen("BANG_TAY", 0)
      Appearance <- "BM_MANU"
   IOField "I/O field_3" at 360,556 size 75x36; FormatPattern s99999
      ProcessValue <- "DEM_CB1"
   IOField "I/O field_4" at 662,552 size 75x36; FormatPattern s99999
      ProcessValue <- "DEM_CB2"
   SymbolLibrary "Symbol library_20" at 349,340 size 45x26
      Appearance <- "M_CB_DAY"
   SymbolLibrary "Symbol library_21" at 939,457 size 29x65
      Appearance <- "M_CB3"
   TextField "Text field_17" at 1149,484 size 56x27; Text 'CB 1:'
   TextField "Text field_18" at 1293,484 size 47x27; Text '[SP]'
   IOField "I/O field_1" at 1209,481 size 84x37; FormatPattern s99999
      ProcessValue <- "DEM_CB1"
   TextField "Text field_19" at 1149,526 size 56x27; Text 'CB 2:'
   TextField "Text field_21" at 1293,526 size 47x27; Text '[SP]'
   IOField "I/O field_2" at 1209,523 size 84x37; FormatPattern s99999
      ProcessValue <- "DEM_CB2"
   TextField "Text field_22" at 1149,568 size 56x27; Text 'CB 3:'
   TextField "Text field_23" at 1293,568 size 47x27; Text '[SP]'
   IOField "I/O field_5" at 1209,565 size 84x37; FormatPattern s99999
      ProcessValue <- "DEM_CB3"
   IOField "I/O field_6" at 913,551 size 75x36; FormatPattern s99999
      ProcessValue <- "DEM_CB3"
   Button "Button_5" at 1152,322 size 88x40; TextOff 'ON'
      on Press: SetBit("BM_SIMULATION")
      Appearance <- "BM_SIMULATION"
   Button "Button_7" at 1152,368 size 88x40; TextOff 'OFF'
      on Press: ResetBit("BM_SIMULATION")
   TextField "Text field_26" at 1270,328 size 59x20; Text 'ĐÈN RUN'
   Circle "Circle_2" at 1275,352 size 49x49
      Appearance <- "Q_DEN_LV"
   SymbolLibrary "Symbol library_19" at 920,661 size 109x52
   SymbolLibrary "Symbol library_22" at 552,661 size 109x52
   SymbolLibrary "Symbol library_23" at 152,661 size 109x45
   Button "Button_6" at 1134,620 size 225x41; TextOff 'EXIT RUNTIME'
      on Press: StopRuntime(0)
   Group "Group_2" at 397,365 size 85x23
   Group "Group_3" at 695,363 size 85x23
   Group "Group_4" at 757,294 size 92x21
   Rectangle "Rectangle_8" at 722,298 size 37x18
      Visibility <- "Q_XL_DAY_NAP"
   Group "Group_5" at 832,295 size 92x21
   TextField "Text field_1" at 123,562 size 205x20; Text 'ĐỘNG CƠ BĂNG CHUYỀN'
   TextField "Text field_2" at 435,551 size 149x20; Text 'XL CHẶN CHAI 1'
   TextField "Text field_3" at 457,572 size 84x20; Text 'XL_CC_1'
   TextField "Text field_4" at 388,526 size 68x22; Text 'CB_1'
   TextField "Text field_5" at 452,301 size 102x20; Text 'XL KẸP 1'
   TextField "Text field_6" at 275,255 size 156x20; Text 'BƠM ĐỊNH LƯỢNG'
   TextField "Text field_7" at 311,278 size 94x20; Text '100ML/S'
   TextField "Text field_8" at 60,190 size 137x20; Text 'BỂ NGUYÊN LIỆU'
   TextField "Text field_9" at 736,550 size 149x20; Text 'XL CHẶN CHAI 2'
   TextField "Text field_10" at 758,571 size 84x20; Text 'XL_CC_2'
   TextField "Text field_11" at 682,525 size 68x22; Text 'CB_2'
   TextField "Text field_12" at 761,339 size 102x20; Text 'XL KẸP 2'
   TextField "Text field_13" at 856,270 size 115x20; Text 'XL ĐẨY NẮP'
   TextField "Text field_14" at 1149,84 size 195x72; Text 'BẢNG ĐIỂU KHIỂN'
   TextField "Text field_20" at 320,319 size 85x20; Text 'CB ĐẦY'
   TextField "Text field_16" at 932,522 size 75x22; Text 'CB_3'
   TextField "Text field_15" at 1155,419 size 174x66; Text 'ĐẾM SẢN PHẨM'
   TextField "Text field_25" at 1149,254 size 202x68; Text 'CHẾ ĐỘ MÔ PHỎNG'
   TextField "Text field_24" at 675,195 size 113x20; Text 'XL DẬP NẮP'
   SymbolLibrary "Symbol library_7" at 395,461 size 29x65
      Appearance <- "M_CB1"
   SymbolLibrary "Symbol library_17" at 420,353 size 39x92
      Visibility <- "BIT_CHAI_MOVE_DOAN_2"
      HorizontalMovement <- "SIMU_DOAN_2"
   SymbolLibrary "Symbol library_24" at 420,353 size 39x92
      Visibility <- "SIMU_CHAI_DANG_ROT"
   Group "Group_1" at 718,346 size 39x102
      HorizontalMovement <- "SIMU_DOAN_3"
   Group "Group_6" at 718,346 size 39x102
   SymbolLibrary "Symbol library_18" at 718,356 size 39x92
      Visibility <- "BIT_CHAI_MOVE_DOAN_3"
   Rectangle "Rectangle_13" at 719,346 size 37x18
      Visibility <- "BIT_CHAI_MOVE_DOAN_3"
   Rectangle "Rectangle_25" at 397,365 size 32x23
      Visibility <- "Q_XLK1"
   Rectangle "Rectangle_26" at 450,365 size 32x23
      Visibility <- "Q_XLK1"
   Rectangle "Rectangle_27" at 695,363 size 32x23
      Visibility <- "Q_XLK2"
   Rectangle "Rectangle_28" at 748,363 size 32x23
      Visibility <- "Q_XLK2"
   Rectangle "Rectangle_29" at 757,294 size 23x21
      Visibility <- "Q_XL_DAY_NAP"
   Rectangle "Rectangle_30" at 779,298 size 70x14
      Visibility <- "Q_XL_DAY_NAP"
   Rectangle "Rectangle_9" at 832,295 size 23x21
      Visibility <- "Q_XL_DAY_NAP"
   Rectangle "Rectangle_31" at 854,299 size 70x14
      Visibility <- "Q_XL_DAY_NAP"
   SymbolLibrary "Symbol library_25" at 718,356 size 39x92
      Visibility <- "SIMU_CHAI_DANG_DONG_NAP"
   Rectangle "Rectangle_32" at 719,346 size 37x18
      Visibility <- "SIMU_CHAI_DANG_DONG_NAP"
*)